Universal Robots PolyScope program: sockets.urp

Program sockets (installation=default directory=/ursim/programs createdIn=5.17.3 lastSavedIn=5.20.0 robotSerialNumber=20195599999)
Calibrated DH parameters: a=[0, -0.425, -0.3922, 0, 0, 0]; d=[0.1625, 0, 0, 0.1333, 0.0997, 0.0996]; alpha=[1.570796, 0, 0, 1.570796, -1.570796, 0]; deltaTheta=[0, 0, 0, 0, 0, 0]
InitVariablesNode
BeforeStart
  Script file /ursim/programs/functions.script
    | socket="s1"
    | len=2
    | 
    | def operacio(mode, currentWidht):
    | 	socket_send_byte(mode ,socket)
    | 	socket_send_byte(currentWidht, socket)
    | 	return socket_read_byte_list(len, socket, 2)
    | end
    | 
    | def open(data, targetWidht):
    | 	currentWidht=data[1]
    | 	while(currentWidht<targetWidht):
    | 		data=operacio(1, currentWidht)
    | 		currentWidht=data[1]
    | 	end
    | 	data=operacio(0, currentWidht)
    | 	return data
    | end
    | 
    | def close(data, targetWidht):
    | 	currentWidht=data[1]
    | 	while(currentWidht>targetWidht):
    | 		data=operacio(2, currentWidht)
    | 		currentWidht=data[1]
    | 	end
    | 	data=operacio(0, currentWidht)
    | 	return data
    | end
  initial_pose := get_actual_tcp_pose()
  ip := "172.23.5.109"
  socket := socket_open(ip, 5858, "s1")
  Loop While (checkContinuously=false) expression=socket≟ False
    socket := socket_open(ip, 5858,"s1")
Robot Program (runOnlyOnce=false)
  data := socket_read_byte_list(2, "s1", 4)
  Loop While (checkContinuously=false) expression=True
    data := close(25, data)
    data := open(42, data)
